INTERFACE I_BaseString

METHOD GetString : STRING
VAR_INPUT
	
END_VAR
END_METHOD

END_INTERFACE

(* stored: Version 1.1.0.1, ProductVersion 3.1.4024.3
   Itf I_BaseString: Id {4b6fe35d-e7c6-418c-8b42-5b4a18d359b4}
   Method GetString: Id {b638e8ac-f10c-4091-b19e-fb9afc817c1e} *)
